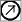
VISUALIZATION VISU_M1Figure_Gauge  // 22x22
    Ellipse (0,0 20x20)
    Line (6,14) (14,6)
    Line (14,12) (14,5)
    Line (15,6) (8,6)
END_VISUALIZATION

(* stored: Version 1.1.0.1, ProductVersion 3.1.4019.2
   Visu VISU_M1Figure_Gauge: Id {5145ba8d-0196-4c6b-a595-05fb93af2550} *)
